// TIA Portal V17 export
// export: Created 2023-04-07T09:30:33.5754766Z, ExportSetting WithDefaults, DisplayName Totally Integrated Automation Portal, DisplayVersion V17 Update 4, DisplayName TIA Portal Openness, DisplayVersion V17 Update 4, DisplayName TIA Portal Version Control Interface, DisplayVersion V17, DisplayName STEP 7 Professional, DisplayVersion V17 Update 4, DisplayName STEP 7 Safety, DisplayVersion V17, DisplayName WinCC Professional, DisplayVersion V17 Update 4
FUNCTION "PCS R (S)_1" : Void   // FC46, LAD
TITLE = ModBus TCP for PCS Power Electronics
{ S7_Optimized_Access := 'TRUE' }
VERSION : 0.1
// stored: AutoNumber true, IsIECCheckEnabled false, SetENOAutomatically false, UDAEnableTagReadback false
   VAR_TEMP
      rVac : Real;
   END_VAR
   VAR_TEMP   // added for the SCL form of the ladder/FBD networks
      _w1 : Bool;
   END_VAR
BEGIN

REGION Network 1: Function Modbus Client
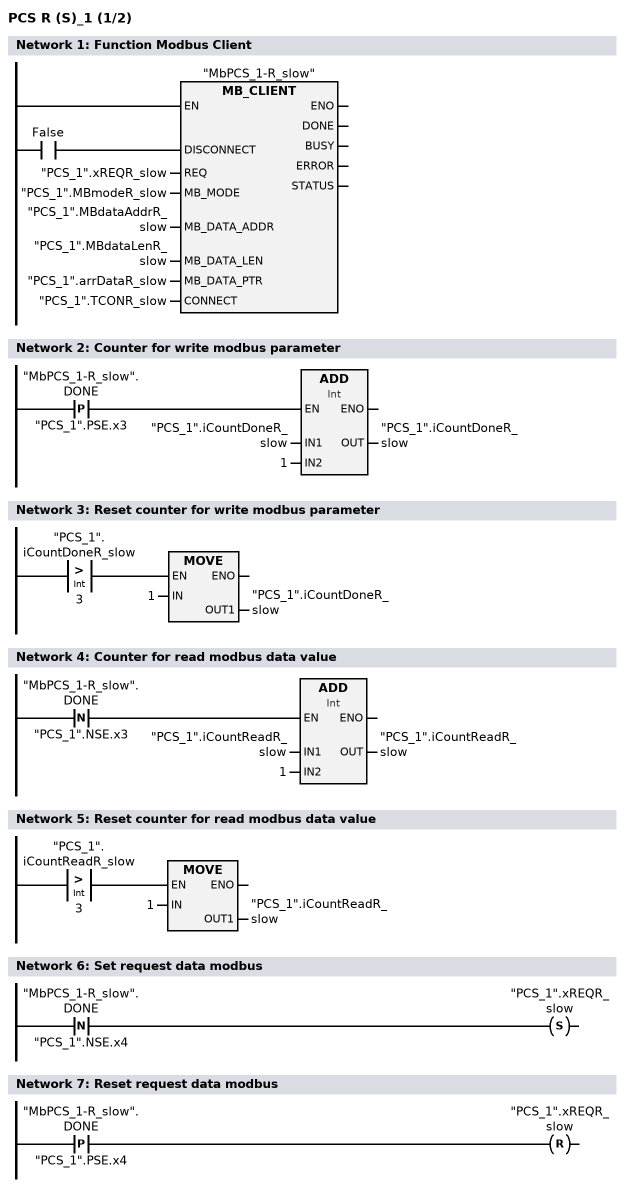
   RUNG wire#powerrail
      "MbPCS_1-R_slow".MB_CLIENT(DISCONNECT := wire#w1, REQ := "PCS_1".xREQR_slow, MB_MODE := "PCS_1".MBmodeR_slow, MB_DATA_ADDR := "PCS_1".MBdataAddrR_slow, MB_DATA_LEN := "PCS_1".MBdataLenR_slow, MB_DATA_PTR := "PCS_1".arrDataR_slow, CONNECT := "PCS_1".TCONR_slow, DONE =>, BUSY =>, ERROR =>, STATUS =>)
   END_RUNG
   RUNG wire#powerrail
      Contact( False )
   END_RUNG wire#w1
   // the same network as SCL:
   "MbPCS_1-R_slow"(DISCONNECT := False,   // MB_CLIENT
                    REQ := "PCS_1".xREQR_slow,
                    MB_MODE := "PCS_1".MBmodeR_slow,
                    MB_DATA_ADDR := "PCS_1".MBdataAddrR_slow,
                    MB_DATA_LEN := "PCS_1".MBdataLenR_slow,
                    MB_DATA_PTR := "PCS_1".arrDataR_slow,
                    CONNECT := "PCS_1".TCONR_slow);
END_REGION

REGION Network 2: Counter for write modbus parameter
   RUNG wire#powerrail
      P_Contact(operand := "MbPCS_1-R_slow".DONE, bit := "PCS_1".PSE.x3)
      { S7_Templates := "SrcType := Int" } Add(in1 := "PCS_1".iCountDoneR_slow, in2 := 1, out => "PCS_1".iCountDoneR_slow)
   END_RUNG
   // the same network as SCL:
   #_w1 := "MbPCS_1-R_slow".DONE AND NOT "PCS_1".PSE.x3;   // rising edge of "MbPCS_1-R_slow".DONE
   "PCS_1".PSE.x3 := "MbPCS_1-R_slow".DONE;
   IF #_w1 THEN "PCS_1".iCountDoneR_slow := "PCS_1".iCountDoneR_slow + 1; END_IF;
END_REGION

REGION Network 3: Reset counter for write modbus parameter
   RUNG wire#powerrail
      { S7_Templates := "SrcType := Int" } GT_Contact(in1 := "PCS_1".iCountDoneR_slow, in2 := 3)
      Move(in := 1, out1 => "PCS_1".iCountDoneR_slow)
   END_RUNG
   // the same network as SCL:
   IF "PCS_1".iCountDoneR_slow > 3 THEN "PCS_1".iCountDoneR_slow := 1; END_IF;
END_REGION

REGION Network 4: Counter for read modbus data value
   RUNG wire#powerrail
      N_Contact(operand := "MbPCS_1-R_slow".DONE, bit := "PCS_1".NSE.x3)
      { S7_Templates := "SrcType := Int" } Add(in1 := "PCS_1".iCountReadR_slow, in2 := 1, out => "PCS_1".iCountReadR_slow)
   END_RUNG
   // the same network as SCL:
   #_w1 := NOT "MbPCS_1-R_slow".DONE AND "PCS_1".NSE.x3;   // falling edge of "MbPCS_1-R_slow".DONE
   "PCS_1".NSE.x3 := "MbPCS_1-R_slow".DONE;
   IF #_w1 THEN "PCS_1".iCountReadR_slow := "PCS_1".iCountReadR_slow + 1; END_IF;
END_REGION

REGION Network 5: Reset counter for read modbus data value
   RUNG wire#powerrail
      { S7_Templates := "SrcType := Int" } GT_Contact(in1 := "PCS_1".iCountReadR_slow, in2 := 3)
      Move(in := 1, out1 => "PCS_1".iCountReadR_slow)
   END_RUNG
   // the same network as SCL:
   IF "PCS_1".iCountReadR_slow > 3 THEN "PCS_1".iCountReadR_slow := 1; END_IF;
END_REGION

REGION Network 6: Set request data modbus
   RUNG wire#powerrail
      N_Contact(operand := "MbPCS_1-R_slow".DONE, bit := "PCS_1".NSE.x4)
      S_Coil( "PCS_1".xREQR_slow )
   END_RUNG
   // the same network as SCL:
   #_w1 := NOT "MbPCS_1-R_slow".DONE AND "PCS_1".NSE.x4;   // falling edge of "MbPCS_1-R_slow".DONE
   "PCS_1".NSE.x4 := "MbPCS_1-R_slow".DONE;
   IF #_w1 THEN "PCS_1".xREQR_slow := TRUE; END_IF;
END_REGION

REGION Network 7: Reset request data modbus
   RUNG wire#powerrail
      P_Contact(operand := "MbPCS_1-R_slow".DONE, bit := "PCS_1".PSE.x4)
      R_Coil( "PCS_1".xREQR_slow )
   END_RUNG
   // the same network as SCL:
   #_w1 := "MbPCS_1-R_slow".DONE AND NOT "PCS_1".PSE.x4;   // rising edge of "MbPCS_1-R_slow".DONE
   "PCS_1".PSE.x4 := "MbPCS_1-R_slow".DONE;
   IF #_w1 THEN "PCS_1".xREQR_slow := FALSE; END_IF;
END_REGION

REGION Network 9: Write RW_Block1 parameter
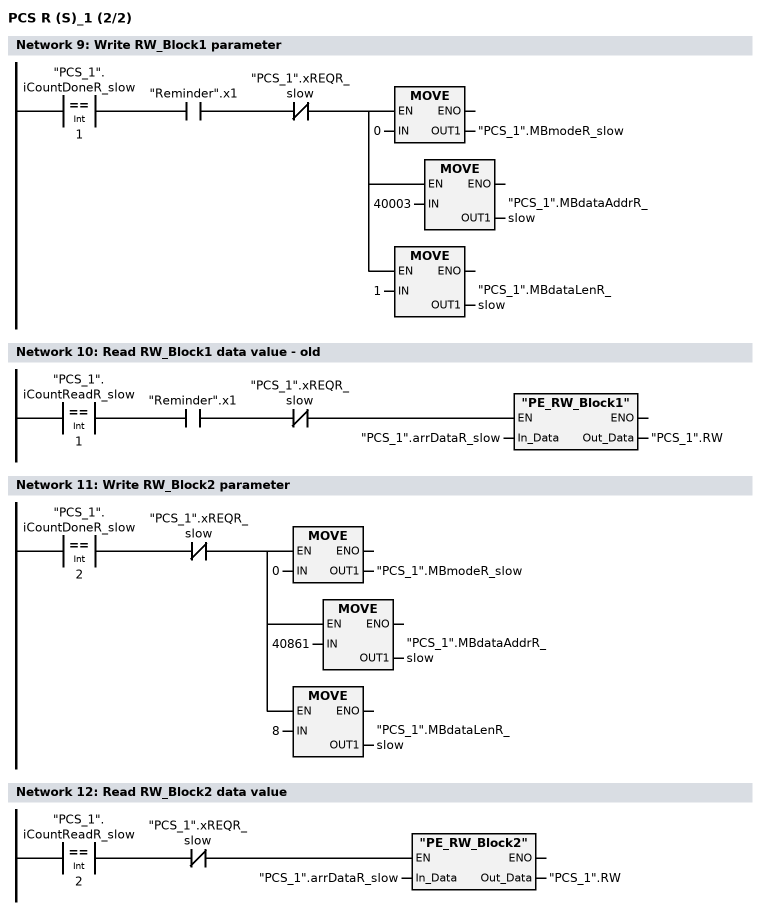
   RUNG wire#powerrail
      { S7_Templates := "SrcType := Int" } EQ_Contact(in1 := "PCS_1".iCountDoneR_slow, in2 := 1)
      Contact( "Reminder".x1 )
      I_Contact( "PCS_1".xREQR_slow )
      wire#w1
      Move(in := 0, out1 => "PCS_1".MBmodeR_slow)
   END_RUNG
   RUNG wire#w1
      Move(in := 40003, out1 => "PCS_1".MBdataAddrR_slow)
   END_RUNG
   RUNG wire#w1
      Move(in := 1, out1 => "PCS_1".MBdataLenR_slow)
   END_RUNG
   // the same network as SCL:
   IF ("PCS_1".iCountDoneR_slow = 1) AND "Reminder".x1 AND NOT "PCS_1".xREQR_slow THEN
       "PCS_1".MBmodeR_slow := 0;
       "PCS_1".MBdataAddrR_slow := 40003;
       "PCS_1".MBdataLenR_slow := 1;
   END_IF;
END_REGION

REGION Network 10: Read RW_Block1 data value - old
   RUNG wire#powerrail
      { S7_Templates := "SrcType := Int" } EQ_Contact(in1 := "PCS_1".iCountReadR_slow, in2 := 1)
      Contact( "Reminder".x1 )
      I_Contact( "PCS_1".xREQR_slow )
      "PE_RW_Block1"(In_Data := "PCS_1".arrDataR_slow, Out_Data => "PCS_1".RW)
   END_RUNG
   // the same network as SCL:
   IF ("PCS_1".iCountReadR_slow = 1) AND "Reminder".x1 AND NOT "PCS_1".xREQR_slow THEN
       "PE_RW_Block1"(In_Data := "PCS_1".arrDataR_slow, Out_Data => "PCS_1".RW);
   END_IF;
END_REGION

REGION Network 11: Write RW_Block2 parameter
   RUNG wire#powerrail
      { S7_Templates := "SrcType := Int" } EQ_Contact(in1 := "PCS_1".iCountDoneR_slow, in2 := 2)
      I_Contact( "PCS_1".xREQR_slow )
      wire#w1
      Move(in := 0, out1 => "PCS_1".MBmodeR_slow)
   END_RUNG
   RUNG wire#w1
      Move(in := 40861, out1 => "PCS_1".MBdataAddrR_slow)
   END_RUNG
   RUNG wire#w1
      Move(in := 8, out1 => "PCS_1".MBdataLenR_slow)
   END_RUNG
   // the same network as SCL:
   IF ("PCS_1".iCountDoneR_slow = 2) AND NOT "PCS_1".xREQR_slow THEN
       "PCS_1".MBmodeR_slow := 0;
       "PCS_1".MBdataAddrR_slow := 40861;
       "PCS_1".MBdataLenR_slow := 8;
   END_IF;
END_REGION

REGION Network 12: Read RW_Block2 data value
   RUNG wire#powerrail
      { S7_Templates := "SrcType := Int" } EQ_Contact(in1 := "PCS_1".iCountReadR_slow, in2 := 2)
      I_Contact( "PCS_1".xREQR_slow )
      "PE_RW_Block2"(In_Data := "PCS_1".arrDataR_slow, Out_Data => "PCS_1".RW)
   END_RUNG
   // the same network as SCL:
   IF ("PCS_1".iCountReadR_slow = 2) AND NOT "PCS_1".xREQR_slow THEN
       "PE_RW_Block2"(In_Data := "PCS_1".arrDataR_slow, Out_Data => "PCS_1".RW);
   END_IF;
END_REGION
END_FUNCTION
